// TIA Portal V20 export
VAR_GLOBAL   // PLC tag table "ConvConstantEmptyLine"
END_VAR
VAR_GLOBAL CONSTANT   // user constants
   minEmptyLine : Int := 2001;
   maxEmptyLine : Int := 2109;
   "J1.1.1" : Int := 2001;   // J1.1.1
   "J1.1.2" : Int := 2002;   // J1.1.2
   "J1.1.3" : Int := 2003;   // J1.1.3
   "J1.1.4" : Int := 2004;   // J1.1.4
   "J1.1.5" : Int := 2005;   // J1.1.5
   "J1.1.6" : Int := 2006;   // J1.1.6
   "J1.1.7" : Int := 2007;   // J1.1.7
   "J1.1.8" : Int := 2008;   // J1.1.8
   "J1.1.9" : Int := 2009;   // J1.1.9
   "J1.1.10" : Int := 2010;   // J1.1.10
   "J1.1.11" : Int := 2011;   // J1.1.11
   "J1.1.12" : Int := 2012;   // J1.1.12
   "J1.1.13" : Int := 2013;   // J1.1.13
   "J1.1.14" : Int := 2014;   // J1.1.14
   "J1.1.15" : Int := 2015;   // J1.1.15
   "J1.2.1" : Int := 2016;   // J1.2.1
   "J1.2.2" : Int := 2017;   // J1.2.2
   "J1.2.3" : Int := 2018;   // J1.2.3 Staright for Merger1
   "J2.1.1" : Int := 2019;   // J2.1.1
   "J2.1.2" : Int := 2020;   // J2.1.2
   "J2.1.3" : Int := 2021;   // J2.1.3
   "J2.1.4" : Int := 2022;   // J2.1.4
   "J2.1.5" : Int := 2023;   // J2.1.5
   "J2.1.6" : Int := 2024;   // J2.1.6
   "J2.1.7" : Int := 2025;   // J2.1.7
   "J2.1.8" : Int := 2026;   // J2.1.8
   "J2.1.9" : Int := 2027;   // J2.1.9
   "J2.1.10" : Int := 2028;   // J2.1.10
   "J2.1.11" : Int := 2029;   // J2.1.11
   "J2.1.12" : Int := 2030;   // J2.1.12
   "J2.1.13" : Int := 2031;   // J2.1.13
   "J2.1.14" : Int := 2032;   // J2.1.14
   "J2.1.15" : Int := 2033;   // J2.1.15
   "J2.2.1" : Int := 2034;   // J2.2.1
   "J2.2.2" : Int := 2035;   // J2.2.2
   "J2.3.1" : Int := 2036;   // J2.3.1
   "J2.4.1" : Int := 2037;   // J2.4.1 Arm for Merger1
   "J1.2.4" : Int := 2038;   // J1.2.4 Merger 1
   "J1.2.5" : Int := 2039;   // J1.2.5
   "J1.3.1" : Int := 2040;   // J1.3.1
   "J1.3.2" : Int := 2041;   // J1.3.2
   "J1.4.1" : Int := 2042;   // J1.4.1
   "J1.4.2" : Int := 2043;   // J1.4.2
   "J1.4.3" : Int := 2044;   // J1.4.3
   "J1.4.4" : Int := 2045;   // J1.4.4
   "J1.4.5" : Int := 2046;   // J1.4.5
   "J1.4.6" : Int := 2047;   // J1.4.6
   "J1.4.7" : Int := 2048;   // J1.4.7
   "J1.5.1" : Int := 2049;   // J1.5.1
   "J1.5.2" : Int := 2050;   // J1.5.2
   "J1.5.3" : Int := 2051;   // J1.5.3
   "J1.5.4" : Int := 2052;   // J1.5.4
   "J1.7.1" : Int := 2053;   // J1.7.1 (Go straight )
   "J1.7.2" : Int := 2054;   // J1.7.2
   "J1.8.1" : Int := 2055;   // J1.8.1
   "J1.8.2" : Int := 2056;   // J1.8.2
   "J1.9.1" : Int := 2057;   // J1.9.1
   "J1.10.1" : Int := 2058;   // J1.10.1
   "J1.11.1" : Int := 2059;   // J1.11.1
   "J1.11.2" : Int := 2060;   // J1.11.2
   "J1.11.3" : Int := 2061;   // J1.11.3
   "J1.11.4" : Int := 2062;   // J1.11.4
   "J1.11.5" : Int := 2063;   // J1.11.5
   "J1.11.6" : Int := 2064;   // J1.11.6
   "J1.11.7" : Int := 2065;   // J1.11.7
   "J1.11.8" : Int := 2066;   // J1.11.8
   "J1.11.9" : Int := 2067;   // J1.11.9
   "J1.11.10" : Int := 2068;   // J1.11.10
   "J1.11.11" : Int := 2069;   // J1.11.11
   "J1.11.12" : Int := 2070;   // J1.11.12
   "J1.11.13" : Int := 2071;   // J1.11.13
   "K1.1.1" : Int := 2072;   // K1.1.1 (Go Left)
   "K1.2.1" : Int := 2073;   // K1.2.1
   "K1.3.1" : Int := 2074;   // K1.3.1
   "K1.4.1" : Int := 2075;   // K1.4.1
   "K1.4.2" : Int := 2076;   // K1.4.2
   "K1.4.3" : Int := 2077;   // K1.4.3
   "K1.4.4" : Int := 2078;   // K1.4.4
   "K1.4.5" : Int := 2079;   // K1.4.5
   "K1.4.6" : Int := 2080;   // K1.4.6
   "K1.4.7" : Int := 2081;   // K1.4.7
   "K1.4.8" : Int := 2082;   // K1.4.8
   "K1.4.9" : Int := 2083;   // K1.4.9
   "K1.4.10" : Int := 2084;   // K1.4.10
   "K1.5.1" : Int := 2085;   // K1.5.1
   "K1.5.2" : Int := 2086;   // K1.5.2
   "K1.5.3" : Int := 2087;   // K1.5.3
   "K1.5.4" : Int := 2088;   // K1.5.4
   "K1.5.5" : Int := 2089;   // K1.5.5
   "K1.5.6" : Int := 2090;   // K1.5.6
   "K1.5.7" : Int := 2091;   // K1.5.7
   "K1.5.8" : Int := 2092;   // K1.5.8
   "K1.6.1" : Int := 2093;   // K1.6.1
   "K1.6.2" : Int := 2094;   // K1.6.2
   "K1.7.1" : Int := 2095;   // K1.7.1
   "K1.7.2" : Int := 2096;   // K1.7.2
   "K1.8.1" : Int := 2097;   // K1.8.1
   "K1.8.2" : Int := 2098;   // K1.8.2
   "K1.8.3" : Int := 2099;   // K1.8.3
   "K1.9.1" : Int := 2100;   // K1.9.1
   "K1.9.2" : Int := 2101;   // K1.9.2
   "K1.9.3" : Int := 2102;   // K1.9.3
   "K1.9.4" : Int := 2103;   // K1.9.4
   "K1.9.5" : Int := 2104;   // K1.9.5
   "K1.9.6" : Int := 2105;   // K1.9.6
   "K1.9.7" : Int := 2106;   // K1.9.7
   "K1.10.1" : Int := 2107;   // K1.10.1
   "J1.6.1" : Int := 2108;   // Mabs J1.6.1
   "J1.6.2" : Int := 2109;   // Mabs J1.6.2
END_VAR
